(* PLC project SafeLOGIC, BrAutomation SafeDESIGNER  5.24.1.0 *)
(* stored: companyURL http://www.br-automation.com, creationDateTime Fri Nov 28 14:27:20 2025 *)

PROGRAM Main
  VAR  (* added by the conversion: wires and edge detectors of the diagram *)
    _BOOL_TO_SAFEBOOL119_OUT : SAFEBOOL;
  END_VAR

(* FBD diagram, written out as Structured Text *)
(* Function 00 - IO and Parameter *)
(* ModuleOK *)
(* Alarm *)
(* Safety loop *)
xKeepAMM_2s_A9433(sbAMMxxxx := AND_S(AND_S(sbSafeModuleOK_SM101, sbSafeModuleOK_SM102, OR_S(sbSafeModuleOK_SM103, AND_S(NOT_S(PARA_LS_HWHT_Lo_Exist), NOT_S(PARA_PS1_HWHT_Hi_Exist), NOT_S(PARA_PS2_HWHT_Hi_Exist), NOT_S(PARA_PS1_HWHT_Lo_Exist), NOT_S(PARA_PS2_HWHT_Lo_Exist), NOT_S(PARA_TS1_HWHT_Hi_Exist), NOT_S(PARA_TS2_HWHT_Hi_Exist), NOT_S(PARA_FS_HWHT_Lo_Exist))), OR_S(sbSafeModuleOK_SM104, AND_S(NOT_S(PARA_LS_HWLT_Lo_Exist), NOT_S(PARA_PS1_HWLT_Hi_Exist), NOT_S(PARA_PS2_HWLT_Hi_Exist), NOT_S(PARA_PS1_HWLT_Lo_Exist), NOT_S(PARA_PS2_HWLT_Lo_Exist), NOT_S(PARA_TS1_HWLT_Hi_Exist), NOT_S(PARA_TS2_HWLT_Hi_Exist), NOT_S(PARA_FS_HWLT_Lo_Exist))), OR_S(sbSafeModuleOK_SM105, AND_S(NOT_S(PARA_HWcirc_Cust_Exist), NOT_S(PARA_SafetyLoop_A2_Exist)))), AND_S(sbSafeModuleOK_SM201, sbSafeModuleOK_SM202, sbSafeModuleOK_SM203, sbSafeModuleOK_SM204, sbSafeModuleOK_SM205, OR_S(sbSafeModuleOK_SM206, NOT_S(PARA_GT2_Exist)), OR_S(sbSafeModuleOK_SM207, NOT_S(PARA_GT3_Exist)), OR_S(sbSafeModuleOK_SM208, AND_S(NOT_S(PARA_GT3_Exist), NOT_S(PARA_GT4_Exist), NOT_S(PARA_DCGA_Exist))), OR_S(sbSafeModuleOK_SM209, NOT_S(PARA_GT4_Exist)), OR_S(sbSafeModuleOK_SM210, NOT_S(PARA_DCGA_Exist))), AND_S(OR_S(sbSafeModuleOK_SM300, PARA_ERV_Cust_Active), OR_S(sbSafeModuleOK_SM301, PARA_ERV_Cust_Active, AND_S(LT_S(PARA_Nr_ERV_INL_Fan, SAFEDINT#5), LT_S(PARA_Nr_ERV_INL_Fan, SAFEDINT#5), LT_S(PARA_Nr_ERV_INL_Fan, SAFEDINT#5))))));
bAMM_A9433 := xKeepAMM_2s_A9433.bAMMxxxx;
sbF00_OK_SafeModuleOK_ALL := xKeepAMM_2s_A9433.sbSL_OK;
(* RESET *)
_BOOL_TO_SAFEBOOL119_OUT := BOOL_TO_SAFEBOOL(bIN_Reset_sPLC);
xF_TRIG_Reset_SL(CLK := _BOOL_TO_SAFEBOOL119_OUT);
xTP_Reset_Safety_2s(IN := AND_S(xF_TRIG_Reset_SL.Q, sbGasValves_Closed), PT := SAFETIME#2s);
sbReset_SafetyLoop := xTP_Reset_Safety_2s.Q;
(* Release Output *)
xRO_SM102(sbReset_sPLC := _BOOL_TO_SAFEBOOL119_OUT, sbSafeModuleOK_SMxxx := sbSafeModuleOK_SM102, sbSafeOutputOK_01 := sbSafeOutputOK_Rel_Sync_Load, sbSafeOutputOK_02 := sbSafeOutputOK_GCB_RUC, sbSafeOutputOK_03 := sbSafeOutputOK_SF_OK_A, sbSafeOutputOK_04 := sbSafeOutputOK_EmStop);
bRO_SM102 := xRO_SM102.bRO_SMxxx;
xRO_SM205(sbReset_sPLC := _BOOL_TO_SAFEBOOL119_OUT, sbSafeModuleOK_SMxxx := sbSafeModuleOK_SM205, sbSafeOutputOK_01 := sbSafeOutputOK_Rel_GV1a, sbSafeOutputOK_02 := sbSafeOutputOK_Rel_GV1b, sbSafeOutputOK_03 := sbSafeOutputOK_GT1_SafeDev, sbSafeOutputOK_04 := sbSafeOutputOK_SF_OK_M);
bRO_SM205 := xRO_SM205.bRO_SMxxx;
xRO_SM206(sbReset_sPLC := _BOOL_TO_SAFEBOOL119_OUT, sbSafeModuleOK_SMxxx := sbSafeModuleOK_SM206, sbSafeOutputOK_01 := sbSafeOutputOK_Rel_GV2a, sbSafeOutputOK_02 := sbSafeOutputOK_Rel_GV2b, sbSafeOutputOK_03 := sbSafeOutputOK_GT2_SafeDev, sbSafeOutputOK_04 := SAFETRUE);
bRO_SM206 := xRO_SM206.bRO_SMxxx;
xRO_SM207(sbReset_sPLC := _BOOL_TO_SAFEBOOL119_OUT, sbSafeModuleOK_SMxxx := sbSafeModuleOK_SM207, sbSafeOutputOK_01 := sbSafeOutputOK_Rel_GV3a, sbSafeOutputOK_02 := sbSafeOutputOK_Rel_GV3b, sbSafeOutputOK_03 := sbSafeOutputOK_GT3_SafeDev, sbSafeOutputOK_04 := SAFETRUE);
bRO_SM207 := xRO_SM207.bRO_SMxxx;
xRO_SM209(sbReset_sPLC := _BOOL_TO_SAFEBOOL119_OUT, sbSafeModuleOK_SMxxx := sbSafeModuleOK_SM209, sbSafeOutputOK_01 := sbSafeOutputOK_Rel_GV4a, sbSafeOutputOK_02 := sbSafeOutputOK_Rel_GV4b, sbSafeOutputOK_03 := sbSafeOutputOK_GT4_SafeDev, sbSafeOutputOK_04 := SAFETRUE);
bRO_SM209 := xRO_SM209.bRO_SMxxx;
xRO_SM210(sbReset_sPLC := _BOOL_TO_SAFEBOOL119_OUT, sbSafeModuleOK_SMxxx := sbSafeModuleOK_SM210, sbSafeOutputOK_01 := sbSafeOutputOK_Rel_GVa_DCGA, sbSafeOutputOK_02 := sbSafeOutputOK_Rel_GVb_DCGA, sbSafeOutputOK_03 := sbSafeOutputOK_DCGA_SafeDev, sbSafeOutputOK_04 := SAFETRUE);
bRO_SM210 := xRO_SM210.bRO_SMxxx;
(* Engine type *)
sbEngineType6 := AND_S(GT_S(PARA_Eng_Motortype, SAFEDINT#600), LT_S(PARA_Eng_Motortype, SAFEDINT#900));
(* PARAMETER to CPU *)
xPARA_BOOL(sbPARA_01 := PARA_GT2_Exist, sbPARA_02 := PARA_GT3_Exist, sbPARA_03 := PARA_GT4_Exist, sbPARA_04 := PARA_SysPurge_MonActive, sbPARA_05 := PARA_HWcirc_Cust_Exist, sbPARA_06 := PARA_PS_HW_Lo_MuteAcive, sbPARA_07 := PARA_LS_HWHT_Lo_Exist, sbPARA_08 := PARA_PS1_HWHT_Hi_Exist, sbPARA_09 := PARA_PS2_HWHT_Hi_Exist, sbPARA_10 := PARA_PS1_HWHT_Lo_Exist, sbPARA_11 := PARA_PS2_HWHT_Lo_Exist, sbPARA_12 := PARA_TS1_HWHT_Hi_Exist, sbPARA_13 := PARA_TS2_HWHT_Hi_Exist, sbPARA_14 := PARA_FS_HWHT_Lo_Exist, sbPARA_15 := PARA_LS_HWLT_Lo_Exist, sbPARA_16 := PARA_PS1_HWLT_Hi_Exist, sbPARA_17 := PARA_PS2_HWLT_Hi_Exist, sbPARA_18 := PARA_PS1_HWLT_Lo_Exist, sbPARA_19 := PARA_PS2_HWLT_Lo_Exist, sbPARA_20 := PARA_TS1_HWLT_Hi_Exist, sbPARA_21 := PARA_TS2_HWLT_Hi_Exist, sbPARA_22 := PARA_FS_HWLT_Lo_Exist, sbPARA_23 := PARA_Pr_EG_sMonActive, sbPARA_24 := PARA_SafetyLoop_A2_Exist, sbPARA_25 := PARA_DCGA_Exist, sbPARA_26 := PARA_ERV_Cust_Active, sbPARA_27 := PARA_ERV_ColdCountry_Active, sbPARA_28 := PARA_ER_Door_MonActive);
bOUT_PARA_GT2_Exist := xPARA_BOOL.bOUT_PARA_01;
bOUT_PARA_GT3_Exist := xPARA_BOOL.bOUT_PARA_02;
bOUT_PARA_GT4_Exist := xPARA_BOOL.bOUT_PARA_03;
bOUT_PARA_SysPurge_MonActive := xPARA_BOOL.bOUT_PARA_04;
bOUT_PARA_HWcirc_Cust_Exist := xPARA_BOOL.bOUT_PARA_05;
bOUT_PARA_PS_HW_Lo_MuteAcive := xPARA_BOOL.bOUT_PARA_06;
bOUT_PARA_LS_HWHT_Lo_Exist := xPARA_BOOL.bOUT_PARA_07;
bOUT_PARA_PS1_HWHT_Hi_Exist := xPARA_BOOL.bOUT_PARA_08;
bOUT_PARA_PS2_HWHT_Hi_Exist := xPARA_BOOL.bOUT_PARA_09;
bOUT_PARA_PS1_HWHT_Lo_Exist := xPARA_BOOL.bOUT_PARA_10;
bOUT_PARA_PS2_HWHT_Lo_Exist := xPARA_BOOL.bOUT_PARA_11;
bOUT_PARA_TS1_HWHT_Hi_Exist := xPARA_BOOL.bOUT_PARA_12;
bOUT_PARA_TS2_HWHT_Hi_Exist := xPARA_BOOL.bOUT_PARA_13;
bOUT_PARA_FS_HWHT_Lo_Exist := xPARA_BOOL.bOUT_PARA_14;
bOUT_PARA_LS_HWLT_Lo_Exist := xPARA_BOOL.bOUT_PARA_15;
bOUT_PARA_PS1_HWLT_Hi_Exist := xPARA_BOOL.bOUT_PARA_16;
bOUT_PARA_PS2_HWLT_Hi_Exist := xPARA_BOOL.bOUT_PARA_17;
bOUT_PARA_PS1_HWLT_Lo_Exist := xPARA_BOOL.bOUT_PARA_18;
bOUT_PARA_PS2_HWLT_Lo_Exist := xPARA_BOOL.bOUT_PARA_19;
bOUT_PARA_TS1_HWLT_Hi_Exist := xPARA_BOOL.bOUT_PARA_20;
bOUT_PARA_TS2_HWLT_Hi_Exist := xPARA_BOOL.bOUT_PARA_21;
bOUT_PARA_FS_HWLT_Lo_Exist := xPARA_BOOL.bOUT_PARA_22;
bOUT_PARA_Pr_EG_sMonActive := xPARA_BOOL.bOUT_PARA_23;
bOUT_PARA_SafetyLoop_A2_Exist := xPARA_BOOL.bOUT_PARA_24;
bOUT_PARA_DCGA_Exist := xPARA_BOOL.bOUT_PARA_25;
bOUT_PARA_ERV_Cust_Active := xPARA_BOOL.bOUT_PARA_26;
bOUT_PARA_ERV_ColdCountry_Act := xPARA_BOOL.bOUT_PARA_27;
bOUT_PARA_ER_Door_MonActive := xPARA_BOOL.bOUT_PARA_28;
xPARA_INT(sPARA_01 := PARA_N_EngNom, sPARA_02 := PARA_N_EngAct_HiHi_Diff, sPARA_03 := PARA_N_Pr_EO_LoLo_Lim1, sPARA_04 := PARA_N_Pr_EO_LoLo_Lim2, sPARA_05 := PARA_Pr_EO_LoLo_LimN1, sPARA_06 := PARA_Pr_EO_LoLo_LimN2, sPARA_07 := PARA_Pr_EO_Diff_EngStop, sPARA_08 := PARA_Pr_EO_HiHi_EngStop, sPARA_09 := PARA_Pr_EO_HiHi_Diff, sPARA_10 := PARA_Pr_EO_HiHi_Check, sPARA_11 := PARA_Pr_EOaP_HiHi, sPARA_12 := PARA_Pr_EOaP_Diff_EngStop, sPARA_13 := PARA_Pr_EOaP_HiHi_EngStop, sPARA_14 := PARA_Pr_ECW_LoLo, sPARA_15 := PARA_Pr_ECW_HiHi_Diff, sPARA_16 := PARA_Pr_ECW_HiHi_Check, sPARA_17 := PARA_Pr_ECWaP_HiHi, sPARA_18 := PARA_Eng_Motortype, sPARA_19 := PARA_DPr_ECWP_LoLo, sPARA_20 := PARA_Vol_SysPurge_Stroke, sPARA_21 := PARA_Vol_SysPurge_MinAir, sPARA_22 := PARA_Nr_ERV_INL_Fan, sPARA_23 := PARA_Nr_ERV_INL_Lou, sPARA_24 := PARA_Nr_ERV_OTL_Lou, sPARA_25 := PARA_NrMaxErr_ERV_INL_Fan, sPARA_26 := PARA_NrMaxErr_ERV_INL_Lou, sPARA_27 := PARA_NrMaxErr_ERV_OTL_Lou);
iOUT_PARA_N_EngNom := xPARA_INT.iOUT_PARA_01;
iOUT_PARA_N_EngAct_HiHi_Diff := xPARA_INT.iOUT_PARA_02;
iOUT_PARA_N_Pr_EO_LoLo_Lim1 := xPARA_INT.iOUT_PARA_03;
iOUT_PARA_N_Pr_EO_LoLo_Lim2 := xPARA_INT.iOUT_PARA_04;
iOUT_PARA_Pr_EO_LoLo_LimN1 := xPARA_INT.iOUT_PARA_05;
iOUT_PARA_Pr_EO_LoLo_LimN2 := xPARA_INT.iOUT_PARA_06;
iOUT_PARA_Pr_EO_Diff_EngStop := xPARA_INT.iOUT_PARA_07;
iOUT_PARA_Pr_EO_HiHi_EngStop := xPARA_INT.iOUT_PARA_08;
iOUT_PARA_Pr_EO_HiHi_Diff := xPARA_INT.iOUT_PARA_09;
iOUT_PARA_Pr_EO_HiHi_Check := xPARA_INT.iOUT_PARA_10;
iOUT_PARA_Pr_EOaP_HiHi := xPARA_INT.iOUT_PARA_11;
iOUT_PARA_Pr_EOaP_Diff_EngStop := xPARA_INT.iOUT_PARA_12;
iOUT_PARA_Pr_EOaP_HiHi_EngStop := xPARA_INT.iOUT_PARA_13;
iOUT_PARA_Pr_ECW_LoLo := xPARA_INT.iOUT_PARA_14;
iOUT_PARA_Pr_ECW_HiHi_Diff := xPARA_INT.iOUT_PARA_15;
iOUT_PARA_Pr_ECW_HiHi_Check := xPARA_INT.iOUT_PARA_16;
iOUT_PARA_Pr_ECWaP_HiHi := xPARA_INT.iOUT_PARA_17;
iOUT_PARA_Eng_Motortype := xPARA_INT.iOUT_PARA_18;
iOUT_PARA_DPr_ECWP_LoLo := xPARA_INT.iOUT_PARA_19;
iOUT_PARA_Vol_SysPurge_Stroke := xPARA_INT.iOUT_PARA_20;
iOUT_PARA_Vol_SysPurge_MinAir := xPARA_INT.iOUT_PARA_21;
iOUT_PARA_Nr_ERV_INL_Fan := xPARA_INT.iOUT_PARA_22;
iOUT_PARA_Nr_ERV_INL_Lou := xPARA_INT.iOUT_PARA_23;
iOUT_PARA_Nr_ERV_OTL_Lou := xPARA_INT.iOUT_PARA_24;
iOUT_PARA_NrMaxErr_ERV_INL_Fan := xPARA_INT.iOUT_PARA_25;
iOUT_PARA_NrMaxErr_ERV_INL_Lou := xPARA_INT.iOUT_PARA_26;
iOUT_PARA_NrMaxErr_ERV_OTL_Lou := xPARA_INT.iOUT_PARA_27;
END_PROGRAM
